# EPICS substitutions: EUROTHRM/EUROTHRM-IOC-01App/Db/devEurothrmA08.substitutions
# Note: this file is generated by generate_substitutions.py
file devEurothrm.template {
pattern { P, GAD, LAD, MODBUS_PV, MODBUS_SP, MODBUS_P, MODBUS_I, MODBUS_D, MODBUS_HS, MODBUS_LS, MODBUS_AT, MODBUS_HO, MODBUS_OP }
{ "\$(P)", "0", "8", "7169", "7170", "7174", "7176", "7177", "7279", "7280", "7438", "7198", "7171" }
}
